(*
A broadcastable wrapper for a `DWORD` value. 
*)
FUNCTION_BLOCK DwordArg IMPLEMENTS I_DwordArg
VAR
	_val			: DWORD;
	_bMut			: BOOL := FALSE;
END_VAR

(*
Enables external modification of the internal value.
*)
METHOD AllowMut
_bMut := TRUE;
END_METHOD

(*
Disables external modification of the internal value.
*)
METHOD BlockMut
_bMut := FALSE;
END_METHOD

(*
Reads the internal value.
*)
PROPERTY Get : DWORD
GET
Get := _val;
END_GET
END_PROPERTY

(*
Returns TRUE if the value is mutable.
*)
PROPERTY IsMut : BOOL
GET
IsMut := _bMut;
END_GET
END_PROPERTY

(*
Directly modifies the internal value, bypassing any mutability restrictions.
*)
METHOD OpSet : I_Arg
VAR_INPUT
	newVal		: DWORD;
END_VAR
_val := newVal;
OpSet := THIS^;
END_METHOD

(*
Modifies the internal value.  
Returns:
- `Ok` - Upon successful modification.
- `Error` - If mutability is disabled.
*)
METHOD Set : Result
VAR_INPUT
	newVal		: DWORD;
END_VAR
IF _bMut THEN
	_val := newVal;
	Set := Ok;
ELSE
	Set := Error;
END_IF
END_METHOD

END_FUNCTION_BLOCK

(* stored: Version 1.1.0.1
   POU DwordArg: Id {9659b537-4688-4285-be75-eafd6725a3aa}, SpecialFunc None
   Method AllowMut: Id {0cf9c6db-9ce8-47a7-bbc6-ae648d557fdb}
   Method BlockMut: Id {f644c949-f11c-42c5-8ff6-fb2a912cef31}
   Property Get: Id {cc59ac16-520a-4813-9448-11df56543b41}
   Get Get: Id {51d7a5da-f031-44c4-96c5-7df19b5ffd36}
   Property IsMut: Id {50b98783-86da-419c-b72c-12661f9da5eb}
   Get Get: Id {c33486f9-6bcd-4602-88a7-537f72d5ce2a}
   Method OpSet: Id {16e7d7ba-329c-43eb-9d90-fd60ed245a15}
   Method Set: Id {3d242843-c798-4d26-8320-230dbe6f25b3} *)
